TYPE "A0301_Mach_Sens_Par"
VERSION : 0.1
// Block: A0301_Mach_Sens_Par
   STRUCT
      Tol_Work : Real;
      WorkTime_SensDisable : Time;
   END_STRUCT;

END_TYPE
